// TIA Portal V17 export
// export: Created 2025-03-10T12:16:40.8089346Z, ExportSetting WithDefaults, DisplayName Totally Integrated Automation Portal, DisplayVersion V17 Update 8, DisplayName TIA Portal Openness, DisplayVersion V17 Update 8, DisplayName TIA Portal Version Control Interface, DisplayVersion V17, DisplayName SINAMICS Startdrive Advanced, DisplayVersion V17 SP2, DisplayName SINAMICS Startdrive G110M, G120, G120C, G120D, G120P, G115D, DisplayVersion V17 SP2, DisplayName SINAMICS Startdrive G130, G150, S120, S150, SINAMICS MV, S210, DisplayVersion V17 SP2, DisplayName STEP 7 Professional, DisplayVersion V17 Update 8, DisplayName SINUMERIK ONE STEP 7 Toolbox, DisplayVersion V17 Update 12, DisplayName SINUMERIK 840D sl STEP 7 Toolbox, DisplayVersion V17 Update 12, DisplayName STEP 7 Safety, DisplayVersion V17 Update 6, DisplayName WinCC Advanced, DisplayVersion V17 Update 8
DATA_BLOCK "LTLP_SLDiagnosticCommandDB"   // DB599
{ DB_Accessible_From_OPC_UA := 'FALSE' }
// stored: AutoNumber false, DBAccessibleFromOPCUA false, DBAccessibleFromWebserver true, InstanceOfName LTLP_SLDiagnosticCommand, InstanceOfType FB
"LTLP_SLDiagnosticCommand"
   // VAR_INPUT
   //    RESTART_PLC : Bool;
   //    ENABLE : Bool;
   // END_VAR
   // VAR_OUTPUT
   //    COMMAND : Int;
   //    BUSY : Bool;
   // END_VAR
   // VAR
   //    reserve1ClassicVersion : Array[6..39] of Byte;
   //    offsetAdressForHMI_Command : Int;
   //    offsetAdressForHMI_Record : Int;
   //    offsetAdressForHMI_ActivCommand : Int;
   //    reserve2ClassicVersion : Array[1..6] of Word;
   //    reserveHMI : Byte;
   //    HMIInterfaceOccupied : Byte;
   //    HMICommand : Struct
   //       Command : Int;
   //       Offset : Byte;
   //       IOID : Byte;
   //       Reserve_Adress : Word;
   //       HardwareID : HW_IO;
   //       RecordNumber : Int;
   //       length : UInt;
   //       buffer : Array[1..240] of Byte;
   //    END_STRUCT;
   //    reserve3ClassicVersion : Array[1..6] of Word;
   //    BusyTime : Time;
   //    reclen : Word;
   //    HMIRecord : Struct
   //       valid : Int;
   //       error : DWord;
   //       buffer : Array[1..1024] of Byte;
   //    END_STRUCT;
   //    HMIActivCommand : Struct
   //       Command : Int;
   //       Offset : Byte;
   //       IOID : Byte;
   //       HardwareID : HW_IO;
   //       Reserve_Adress : Word;
   //       RecordNumber : Int;
   //       length : UInt;
   //       function : Int;
   //    END_STRUCT;
   //    ReadWriteDeviceRecord : Array[1..241] of Byte;
   //    ReadDiagnosticDataNew : Bool;
   //    WriteDiagnosticDataNew : Bool;
   //    ReadDiagnosticDataActiv : Bool;
   //    WriteDiagnosticDataActiv : Bool;
   //    ResetDiagnosticDataActiv : Bool;
   //    Command_1 : Bool;
   //    reserve_x6 : Bool;
   //    trigHMIInterfaceOccupied : Bool;
   //    HMIInterfaceOccupiedTime : Time;
   //    ReadDeviceData { S7_SetPoint := 'True'} : RDREC;
   //    WriteDeviceData { S7_SetPoint := 'True'} : WRREC;
   // END_VAR
BEGIN
END_DATA_BLOCK
